FUNCTION_BLOCK SK_MoveUp (* Atomic skill MoveUp (parameters: none); owns its actuator output; uniform skill interface: CALL/DONE/FAILED, unit control, cell sample, status chain, OPC UA facade *)
  (* Standard: 61499-2 *)
  (* Version 2.0, 2026-09-27, Project contributors, Filling cell reference model *)
  PACKAGE fillingcell;
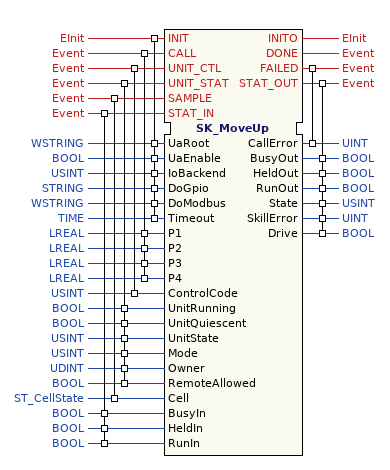
  EVENT_INPUT
    INIT : EInit WITH UaRoot, UaEnable, IoBackend, DoGpio, DoModbus, Timeout;
    CALL WITH P1, P2, P3, P4;
    UNIT_CTL WITH ControlCode;
    UNIT_STAT WITH UnitRunning, UnitQuiescent, UnitState, Mode, Owner, RemoteAllowed;
    SAMPLE WITH Cell;
    STAT_IN WITH BusyIn, HeldIn, RunIn;
  END_EVENT
  EVENT_OUTPUT
    INITO : EInit;
    DONE;
    FAILED WITH CallError;
    STAT_OUT WITH BusyOut, HeldOut, RunOut, State, SkillError, Drive;
  END_EVENT
  VAR_INPUT
    UaRoot : WSTRING;
    UaEnable : BOOL;
    IoBackend : USINT;
    DoGpio : STRING;
    DoModbus : WSTRING;
    Timeout : TIME := T#10s;
    P1 : LREAL;
    P2 : LREAL;
    P3 : LREAL;
    P4 : LREAL;
    ControlCode : USINT;
    UnitRunning : BOOL;
    UnitQuiescent : BOOL;
    UnitState : USINT;
    Mode : USINT;
    Owner : UDINT;
    RemoteAllowed : BOOL;
    Cell : fillingcell::ST_CellState;
    BusyIn : BOOL;
    HeldIn : BOOL := TRUE;
    RunIn : BOOL := TRUE;
  END_VAR
  VAR_OUTPUT
    CallError : UINT;
    BusyOut : BOOL;
    HeldOut : BOOL;
    RunOut : BOOL;
    State : USINT := 4;
    SkillError : UINT;
    Drive : BOOL;
  END_VAR
  FBS
    Gate : fillingcell::SKILL_Gate;
    Pml : fillingcell::SKILL_PackML;
    Logic : fillingcell::SL_MoveUp;
    Wd : iec61499::events::E_DELAY;
    Chain : fillingcell::SKILL_Chain;
    Ua : fillingcell::UA_SkillFacade;
    Out : fillingcell::IO_DO;
  END_FBS
  EVENT_CONNECTIONS
    INIT TO Ua.INIT;
    Ua.INITO TO Out.INIT;
    Out.INITO TO INITO;
    CALL TO Gate.CALL;
    UNIT_CTL TO Gate.UNIT_CTL;
    UNIT_STAT TO Gate.UNIT_STAT;
    Ua.MCMD TO Gate.MCMD;
    Gate.CMD TO Pml.CMD;
    Gate.START TO Logic.CHECK;
    Logic.CHECKED TO Pml.CMD;
    Gate.DONE TO DONE;
    Gate.FAILED TO FAILED;
    Gate.M_ACK TO Ua.M_ACK;
    Gate.M_REJ TO Ua.M_REJ;
    SAMPLE TO Logic.EVAL;
    Logic.COND TO Pml.COND;
    Pml.LATCH TO Logic.LATCH;
    Pml.REJECTED TO Gate.REJ;
    Pml.WD_START TO Wd.START;
    Pml.WD_STOP TO Wd.STOP;
    Wd.EO TO Pml.TIMEOUT;
    Pml.CNF TO Gate.TRACK;
    Pml.CNF TO Chain.REQ;
    Pml.CNF TO Ua.PUB;
    Pml.CNF TO Out.REQ;
    Logic.LATCHED TO Ua.PUB;
    STAT_IN TO Chain.REQ;
    Gate.POKE TO Chain.REQ;
    Chain.CNF TO STAT_OUT;
  END_CONNECTIONS
  DATA_CONNECTIONS
    UaRoot TO Ua.UaRoot;
    UaEnable TO Ua.UaEnable;
    IoBackend TO Out.Backend;
    DoGpio TO Out.GpioName;
    DoModbus TO Out.ModbusId;
    Timeout TO Wd.DT;
    P1 TO Gate.P1;
    P2 TO Gate.P2;
    P3 TO Gate.P3;
    P4 TO Gate.P4;
    ControlCode TO Gate.ControlCode;
    UnitRunning TO Gate.UnitRunning;
    UnitQuiescent TO Gate.UnitQuiescent;
    UnitState TO Gate.UnitState;
    Mode TO Gate.Mode;
    Owner TO Gate.Owner;
    RemoteAllowed TO Gate.RemoteAllowed;
    Ua.Requester TO Gate.Requester;
    Ua.MCode TO Gate.MCode;
    Ua.MP1 TO Gate.MP1;
    Ua.MP2 TO Gate.MP2;
    Ua.MP3 TO Gate.MP3;
    Ua.MP4 TO Gate.MP4;
    Gate.Command TO Pml.Command;
    Gate.PO1 TO Logic.P1;
    Gate.PO2 TO Logic.P2;
    Gate.PO3 TO Logic.P3;
    Gate.PO4 TO Logic.P4;
    Logic.RequiresOK TO Pml.RequiresOK;
    Gate.CallError TO CallError;
    Gate.MErr TO Ua.MErr;
    Cell TO Logic.Cell;
    Logic.EnsuresOK TO Pml.EnsuresOK;
    Logic.InvariantOK TO Pml.InvariantOK;
    Pml.State TO Gate.State;
    Pml.State TO Chain.State;
    Pml.State TO Ua.State;
    Pml.State TO State;
    Pml.ErrorID TO Gate.SkillError;
    Pml.ErrorID TO Ua.ErrorID;
    Pml.ErrorID TO SkillError;
    Pml.Active TO Out.OUT;
    Pml.Active TO Drive;
    Logic.P1L TO Ua.P1;
    Logic.P2L TO Ua.P2;
    Logic.P3L TO Ua.P3;
    Logic.P4L TO Ua.P4;
    BusyIn TO Chain.BusyIn;
    HeldIn TO Chain.HeldIn;
    RunIn TO Chain.RunIn;
    Chain.BusyOut TO BusyOut;
    Chain.HeldOut TO HeldOut;
    Chain.RunOut TO RunOut;
  END_CONNECTIONS
END_FUNCTION_BLOCK
